// TwinCAT 3 PLC project PlcHammer
// Title: PlcHammer
// Company: Vortex.Library
// ProjectVersion: 0.6.0.913
// ProgramVersion: 3.1.4023.0
// libraries:
//   Tc2_Math, * (Beckhoff Automation GmbH)
//   Tc2_Standard, * (Beckhoff Automation GmbH)
//   Tc2_System, * (Beckhoff Automation GmbH)
//   Tc3_Module, * (Beckhoff Automation GmbH)
//   TcoCore, 0.8.1.3 (Vortex.Library)
//   TcoData, 0.8.1.3 (Vortex.Library)
//   TcoDrivesBeckhoff, 0.8.1.3 (Vortex.Library)
//   TcoElements, 0.8.1.3 (Vortex.Library)
//   TcoInspectors, 0.6.0.913 (Vortex.Library)
//   TcoIo, 0.8.1.3 (Vortex.Library)
//   TcoPneumatics, 0.8.1.3 (Vortex.Library)
// project tree:
//   Components/Drive/ DriveSim.TcPOU (not stored), DriveSimMoveAbsoluteTask.TcPOU (not stored), IDrive.TcIO (not stored)
//   DUTs/Enums/ enumColors.TcDUT, enumModes.TcDUT (not stored)
//   DUTs/Structs/CutomLibraries/ VortexComponent.TcDUT
//   DUTs/Structs/GenericStructs/ Car.TcDUT, VariousTypes.TcDUT, Wheel.TcDUT
//   DUTs/Structs/LayoutTests/Border/ BorderLayout.TcDUT, Border_other.TcDUT
//   DUTs/Structs/LayoutTests/GroupBox/ GroupBoxLayout.TcDUT, GroupBox_other.TcDUT
//   DUTs/Structs/LayoutTests/Multiple/ Border_other_other.TcDUT, GroupBox_other_other.TcDUT, Scroll_other_other.TcDUT, Stack_other_other.TcDUT, Tabs_other_other.TcDUT, UniformGrid_other_other.TcDUT, Wrap_other_other.TcDUT
//   DUTs/Structs/LayoutTests/Scroll/ ScrollLayout.TcDUT, Scroll_other.TcDUT
//   DUTs/Structs/LayoutTests/Stack/ StackLayout.TcDUT, Stack_other.TcDUT
//   DUTs/Structs/LayoutTests/Tabs/ TabsLayout.TcDUT (not stored), Tabs_other.TcDUT
//   DUTs/Structs/LayoutTests/UniformGrid/ UniformGridLayout.TcDUT, UniformGrid_other.TcDUT
//   DUTs/Structs/ LayoutTests.TcDUT, RenderIgnoreTests.TcDUT
//   DUTs/Structs/LayoutTests/Wrap/ WrapLayout.TcDUT (not stored), Wrap_other.TcDUT
//   DUTs/Structs/RenderIgnore/ RenderIgnore_basic.TcDUT
//   Misc/Checkers/ Checkers.TcPOU (not stored), AnalogueValueCheck.TcDUT (not stored), eCheckResult.TcDUT (not stored)
//   / PlcTask.TcTTO (not stored)
//   POUs/ AppContext.TcPOU (not stored), TECH_MAIN.TcPOU (not stored)
//   POUs/Data/ ProcessDataManager.TcPOU (not stored), RealValueSimulation.TcPOU (not stored), TechnologicalDataManager.TcPOU (not stored)
//   POUs/Station001/ Station001_Swift.TcPOU (not stored), IO.TcGVL (not stored), Station001.TcPOU, Station001_Components.TcPOU (not stored), Station001_GroundMode.TcPOU (not stored), Station001_AutomatMode.TcPOU (not stored), Station001_ProductionData.TcDUT (not stored), Station001_TechnologicalSettings.TcDUT (not stored)
// real-time tasks:
//   TASK PlcTask: cycle T#10ms, priority 20, ADS port 350
// motion (NC):
//   TASK NC-Task 1 SAF: cycle T#2ms, priority 4, ADS port 501
//   TASK NC-Task 1 SVB: cycle T#10ms, priority 8, ADS port 511
//   AXIS Axis 1 (id 1)
//     OtherSettings: AllowMotionCmdToSlave=true
//     encoder EncType=1
//     drive DrvType=5
//       Analog: TorqueSetpointScale=10, ScaleFactorActTorque=0.1
//       TimeComp: TaskDelayCycles=1
//     controller CtrType=1
//       CtrPara: PriorControlFactor=1
//         Observer: BandWidth=20
// variable links:
//   PlcHammer/PlcHammer Instance <-> NC-Task 1 SAF/Axes/Axis 1
//     PlcTask Inputs/IO.Axis1.NcToPlc <-> Outputs/ToPlc
//     PlcTask Outputs/IO.Axis1.PlcToNc <-> Inputs/FromPlc

// ---- DUTs/Enums/enumColors.TcDUT
{attribute 'qualified_only'}
{attribute 'strict'}
TYPE enumColors :
(
	Red := 0,
	Orange := 1,
	Yellow := 2,
	Green := 3,
	Blue := 4,
	Indigo := 5,
	Violet := 6
);
END_TYPE

// ---- DUTs/Structs/CutomLibraries/VortexComponent.TcDUT
TYPE VortexComponent :
STRUCT
	vortex_bool: BOOL;
	vortex_int: INT;
	vortex_string: STRING;
	vortex_wheel: Wheel;
END_STRUCT
END_TYPE

// ---- DUTs/Structs/GenericStructs/Car.TcDUT
TYPE Car :
STRUCT
	_manufacturer: STRING;
	_model: STRING;
	_manufactured_time: DATE_AND_TIME;
	_ready_for_UK: BOOL;
	_color: enumColors;
	_width: REAL;
	_height: REAL;
	_length: REAL;
	_price: USINT;
END_STRUCT
END_TYPE

// ---- DUTs/Structs/GenericStructs/VariousTypes.TcDUT
TYPE VariousTypes :
STRUCT
	_BOOL_00          : BOOL;
	_INT_00           : INT;
	{attribute addProperty Name "<#_UINT_00 with subrange 69-420#>"}
	_UINT_00          : UINT (69..420);
	_ULINT_00         : ULINT := 18446744073709551615;
	_REAL_00          : REAL := 2.718281828;
	_BYTE_00          : BYTE := 2#00000101;
	_DATE_AND_TIME_00 : DATE_AND_TIME := DT#2000-01-01-00:00:00.01;
	_LTIME_00         : LTIME := LTIME#2D0H45M1S563MS333US880NS;
	{attribute clr [RenderIgnore()]}
	_STRING_00        : STRING;
	_STRING_01        : STRING := 'How are you?';
	_ptString         : POINTER TO STRING := ADR(_STRING_01);
	_eColors_00       : enumColors := enumColors.Red;
END_STRUCT
END_TYPE

// ---- DUTs/Structs/GenericStructs/Wheel.TcDUT
TYPE Wheel :
STRUCT
	_rim_radius: REAL;
	_material: STRING;
	_manufactured_time: DATE_AND_TIME;
END_STRUCT
END_TYPE

// ---- DUTs/Structs/LayoutTests/Border/BorderLayout.TcDUT
{attribute wpf [Container(Layout.Border)]}
TYPE BorderLayout:
STRUCT
	_various_types: VariousTypes;
END_STRUCT
END_TYPE

// ---- DUTs/Structs/LayoutTests/Border/Border_other.TcDUT
{attribute wpf [Container(Layout.Border)]}
TYPE Border_other :
STRUCT
	{attribute wpf [Container(Layout.Stack)]}
	_wheel_stack: Wheel;
	{attribute wpf [Container(Layout.UniformGrid)]}
	_wheel_ug: Wheel;
	{attribute wpf [Container(Layout.Wrap)]}
	_wheel_wrap: Wheel;
	{attribute wpf [Container(Layout.Tabs)]}
	_wheel_tabs: Wheel;
	{attribute wpf [Container(Layout.Border)]}
	_wheel_border: Wheel;
	{attribute wpf [Container(Layout.GroupBox)]}
	_wheel_gb: Wheel;
	{attribute wpf [Container(Layout.Scroll)]}
	_wheel_scroll: Wheel;
END_STRUCT
END_TYPE

// ---- DUTs/Structs/LayoutTests/GroupBox/GroupBoxLayout.TcDUT
TYPE GroupBoxLayout:
STRUCT
	{attribute wpf [Container(Layout.Stack)]}
	{attribute wpf [Group(Layout.GroupBox)]}
	{attribute addProperty Name "<#Various types#>"}
	_vt: VariousTypes;
END_STRUCT
END_TYPE

// ---- DUTs/Structs/LayoutTests/GroupBox/GroupBox_other.TcDUT
{attribute wpf [Container(Layout.GroupBox)]}
TYPE GroupBox_other :
STRUCT
	{attribute wpf [Container(Layout.Stack)]}
	_wheel_stack: Wheel;
	{attribute wpf [Container(Layout.UniformGrid)]}
	_wheel_ug: Wheel;
	{attribute wpf [Container(Layout.Wrap)]}
	_wheel_wrap: Wheel;
//	{attribute wpf [Container(Layout.Tabs)]}
//	_wheel_tabs: Wheel;
	{attribute wpf [Container(Layout.Border)]}
	_wheel_border: Wheel;
	{attribute wpf [Container(Layout.Scroll)]}
	_wheel_scroll: Wheel;
END_STRUCT
END_TYPE

// ---- DUTs/Structs/LayoutTests/Multiple/Border_other_other.TcDUT
{attribute wpf [Container(Layout.Border)]}
TYPE Border_other_other :
STRUCT
	{attribute addProperty Name "<#Stack#>"}
	_stack_other: Stack_other;
	{attribute addProperty Name "<#UniformGrid#>"}
	_uniformGrid_other: UniformGrid_other;
	{attribute addProperty Name "<#Wrap#>"}
	_wrap_other: Wrap_other;
	{attribute addProperty Name "<#Tabs#>"}
	_tabs_other: Tabs_other;
	{attribute addProperty Name "<#Border#>"}
	_border_other: Border_other;
	{attribute addProperty Name "<#GroupBox#>"}
	_groupBox_other: GroupBox_other;
	{attribute addProperty Name "<#Scroll#>"}
	_scroll_other: Scroll_other;
END_STRUCT
END_TYPE

// ---- DUTs/Structs/LayoutTests/Multiple/GroupBox_other_other.TcDUT
{attribute wpf [Container(Layout.GroupBox)]}
TYPE GroupBox_other_other :
STRUCT
	{attribute addProperty Name "<#Stack#>"}
	_stack_other: Stack_other;
	{attribute addProperty Name "<#UniformGrid#>"}
	_uniformGrid_other: UniformGrid_other;
	{attribute addProperty Name "<#Wrap#>"}
	_wrap_other: Wrap_other;
	{attribute addProperty Name "<#Tabs#>"}
	_tabs_other: Tabs_other;
	{attribute addProperty Name "<#Border#>"}
	_border_other: Border_other;
	{attribute addProperty Name "<#GroupBox#>"}
	_groupBox_other: GroupBox_other;
	{attribute addProperty Name "<#Scroll#>"}
	_scroll_other: Scroll_other;
END_STRUCT
END_TYPE

// ---- DUTs/Structs/LayoutTests/Multiple/Scroll_other_other.TcDUT
{attribute wpf [Container(Layout.Scroll)]}
TYPE Scroll_other_other :
STRUCT
	{attribute addProperty Name "<#Stack#>"}
	_stack_other: Stack_other;
	{attribute addProperty Name "<#UniformGrid#>"}
	_uniformGrid_other: UniformGrid_other;
	{attribute addProperty Name "<#Wrap#>"}
	_wrap_other: Wrap_other;
	{attribute addProperty Name "<#Tabs#>"}
	_tabs_other: Tabs_other;
	{attribute addProperty Name "<#Border#>"}
	_border_other: Border_other;
	{attribute addProperty Name "<#GroupBox#>"}
	_groupBox_other: GroupBox_other;
	{attribute addProperty Name "<#Scroll#>"}
	_scroll_other: Scroll_other;
END_STRUCT
END_TYPE

// ---- DUTs/Structs/LayoutTests/Multiple/Stack_other_other.TcDUT
{attribute wpf [Container(Layout.Stack)]}
TYPE Stack_other_other :
STRUCT
	{attribute addProperty Name "<#Stack#>"}
	_stack_other: Stack_other;
	{attribute addProperty Name "<#UniformGrid#>"}
	_uniformGrid_other: UniformGrid_other;
	{attribute addProperty Name "<#Wrap#>"}
	_wrap_other: Wrap_other;
	{attribute addProperty Name "<#Tabs#>"}
	_tabs_other: Tabs_other;
	{attribute addProperty Name "<#Border#>"}
	_border_other: Border_other;
	{attribute addProperty Name "<#GroupBox#>"}
	_groupBox_other: GroupBox_other;
	{attribute addProperty Name "<#Scroll#>"}
	_scroll_other: Scroll_other;
END_STRUCT
END_TYPE

// ---- DUTs/Structs/LayoutTests/Multiple/Tabs_other_other.TcDUT
{attribute wpf [Container(Layout.Tabs)]}
TYPE Tabs_other_other :
STRUCT
	{attribute addProperty Name "<#Stack#>"}
	_stack_other: Stack_other;
	{attribute addProperty Name "<#UniformGrid#>"}
	_uniformGrid_other: UniformGrid_other;
	{attribute addProperty Name "<#Wrap#>"}
	_wrap_other: Wrap_other;
	{attribute addProperty Name "<#Tabs#>"}
	_tabs_other: Tabs_other;
	{attribute addProperty Name "<#Border#>"}
	_border_other: Border_other;
	{attribute addProperty Name "<#GroupBox#>"}
	_groupBox_other: GroupBox_other;
	{attribute addProperty Name "<#Scroll#>"}
	_scroll_other: Scroll_other;
END_STRUCT
END_TYPE

// ---- DUTs/Structs/LayoutTests/Multiple/UniformGrid_other_other.TcDUT
{attribute wpf [Container(Layout.UniformGrid)]}
TYPE UniformGrid_other_other :
STRUCT
	{attribute addProperty Name "<#Stack#>"}
	_stack_other: Stack_other;
	{attribute addProperty Name "<#UniformGrid#>"}
	_uniformGrid_other: UniformGrid_other;
	{attribute addProperty Name "<#Wrap#>"}
	_wrap_other: Wrap_other;
	{attribute addProperty Name "<#Tabs#>"}
	_tabs_other: Tabs_other;
	{attribute addProperty Name "<#Border#>"}
	_border_other: Border_other;
	{attribute addProperty Name "<#GroupBox#>"}
	_groupBox_other: GroupBox_other;
	{attribute addProperty Name "<#Scroll#>"}
	_scroll_other: Scroll_other;
END_STRUCT
END_TYPE

// ---- DUTs/Structs/LayoutTests/Multiple/Wrap_other_other.TcDUT
{attribute wpf [Container(Layout.Wrap)]}
TYPE Wrap_other_other :
STRUCT
	{attribute addProperty Name "<#Stack#>"}
	_stack_other: Stack_other;
	{attribute addProperty Name "<#UniformGrid#>"}
	_uniformGrid_other: UniformGrid_other;
	{attribute addProperty Name "<#Wrap#>"}
	_wrap_other: Wrap_other;
	{attribute addProperty Name "<#Tabs#>"}
	_tabs_other: Tabs_other;
	{attribute addProperty Name "<#Border#>"}
	_border_other: Border_other;
	{attribute addProperty Name "<#GroupBox#>"}
	_groupBox_other: GroupBox_other;
	{attribute addProperty Name "<#Scroll#>"}
	_scroll_other: Scroll_other;
END_STRUCT
END_TYPE

// ---- DUTs/Structs/LayoutTests/Scroll/ScrollLayout.TcDUT
{attribute wpf [Container(Layout.Scroll)]}
TYPE ScrollLayout :
STRUCT
	_vt: VariousTypes;
END_STRUCT
END_TYPE

// ---- DUTs/Structs/LayoutTests/Scroll/Scroll_other.TcDUT
{attribute wpf [Container(Layout.Scroll)]}
TYPE Scroll_other :
STRUCT
	{attribute wpf [Container(Layout.Stack)]}
	_wheel_stack: Wheel;
	{attribute wpf [Container(Layout.UniformGrid)]}
	_wheel_ug: Wheel;
	{attribute wpf [Container(Layout.Wrap)]}
	_wheel_wrap: Wheel;
	{attribute wpf [Container(Layout.Tabs)]}
	_wheel_tabs: Wheel;
	{attribute wpf [Container(Layout.Border)]}
	_wheel_border: Wheel;
	{attribute wpf [Container(Layout.GroupBox)]}
	_wheel_gb: Wheel;
	{attribute wpf [Container(Layout.Scroll)]}
	_wheel_scroll: Wheel;
END_STRUCT
END_TYPE

// ---- DUTs/Structs/LayoutTests/Stack/StackLayout.TcDUT
{attribute wpf [Container(Layout.Stack)]}
TYPE StackLayout:
STRUCT
	_various_types: VariousTypes;
END_STRUCT
END_TYPE

// ---- DUTs/Structs/LayoutTests/Stack/Stack_other.TcDUT
{attribute wpf [Container(Layout.Stack)]}
TYPE Stack_other :
STRUCT
	{attribute wpf [Container(Layout.Stack)]}
	_wheel_stack: Wheel;
	{attribute wpf [Container(Layout.UniformGrid)]}
	_wheel_ug: Wheel;
	{attribute wpf [Container(Layout.Wrap)]}
	_wheel_wrap: Wheel;
	{attribute wpf [Container(Layout.Tabs)]}
	_wheel_tabs: Wheel;
	{attribute wpf [Container(Layout.Border)]}
	_wheel_border: Wheel;
	{attribute wpf [Container(Layout.GroupBox)]}
	_wheel_gb: Wheel;
	{attribute wpf [Container(Layout.Scroll)]}
	_wheel_scroll: Wheel;
END_STRUCT
END_TYPE

// ---- DUTs/Structs/LayoutTests/Tabs/Tabs_other.TcDUT
{attribute wpf [Container(Layout.Tabs)]}
TYPE Tabs_other :
STRUCT
	{attribute addProperty Name "<#Stack#>"}
	{attribute wpf [Container(Layout.Stack)]}
	_wheel_stack: Wheel;
	{attribute addProperty Name "<#UniformGrid#>"}
	{attribute wpf [Container(Layout.UniformGrid)]}
	_wheel_ug: Wheel;
	{attribute addProperty Name "<#Wrap#>"}
	{attribute wpf [Container(Layout.Wrap)]}
	_wheel_wrap: Wheel;
	{attribute addProperty Name "<#Tabs#>"}
	{attribute wpf [Container(Layout.Tabs)]}
	_wheel_tabs: Wheel;
	{attribute addProperty Name "<#Border#>"}
	{attribute wpf [Container(Layout.Border)]}
	_wheel_border: Wheel;
	{attribute addProperty Name "<#GroupBox#>"}
	{attribute wpf [Container(Layout.GroupBox)]}
	_wheel_gb: Wheel;
	{attribute addProperty Name "<#Scroll#>"}
	{attribute wpf [Container(Layout.Scroll)]}
	_wheel_scroll: Wheel;
END_STRUCT
END_TYPE

// ---- DUTs/Structs/LayoutTests/UniformGrid/UniformGridLayout.TcDUT
{attribute wpf [Container(Layout.UniformGrid)]}
TYPE UniformGridLayout:
STRUCT
	_various_types: VariousTypes;
END_STRUCT
END_TYPE

// ---- DUTs/Structs/LayoutTests.TcDUT
TYPE LayoutTests :
STRUCT
	_stackLayout: StackLayout;
	_uniformGridLayout: UniformGridLayout;
	_wrapLayout: WrapLayout;
	_tabsLayout: TabsLayout;
	_borderLayout: BorderLayout;
	_groupBoxLayout: GroupBoxLayout;
	_scrollLayout: ScrollLayout;
	
	// multiple 2nd layer
	_stack_other: Stack_other;
	_uniformGrid_other: UniformGrid_other;
	_wrap_other: Wrap_other;
	_tabs_other: Tabs_other;
	_border_other: Border_other;
	_groupBox_other: GroupBox_other;
	_scroll_other: Scroll_other;
	
	//multiple 3rd layer xddds
	_stack_other_other: Stack_other_other;
	_uniformGrid_other_other: UniformGrid_other_other;
	_wrap_other_other: Wrap_other_other;
	_tabs_other_other: Tabs_other_other;
	_border_other_other: Border_other_other;
	_groupBox_other_other: GroupBox_other_other;
	_scroll_other_other: Scroll_other_other;
END_STRUCT
END_TYPE

// ---- DUTs/Structs/LayoutTests/UniformGrid/UniformGrid_other.TcDUT
{attribute wpf [Container(Layout.UniformGrid)]}
TYPE UniformGrid_other :
STRUCT
	{attribute wpf [Container(Layout.Stack)]}
	_wheel_stack: Wheel;
	{attribute wpf [Container(Layout.UniformGrid)]}
	_wheel_ug: Wheel;
	{attribute wpf [Container(Layout.Wrap)]}
	_wheel_wrap: Wheel;
	{attribute wpf [Container(Layout.Tabs)]}
	_wheel_tabs: Wheel;
	{attribute wpf [Container(Layout.Border)]}
	_wheel_border: Wheel;
	{attribute wpf [Container(Layout.GroupBox)]}
	_wheel_gb: Wheel;
	{attribute wpf [Container(Layout.Scroll)]}
	_wheel_scroll: Wheel;
END_STRUCT
END_TYPE

// ---- DUTs/Structs/LayoutTests/Wrap/Wrap_other.TcDUT
{attribute wpf [Container(Layout.Wrap)]}
TYPE Wrap_other :
STRUCT
	{attribute wpf [Container(Layout.Stack)]}
	_wheel_stack: Wheel;
	{attribute wpf [Container(Layout.UniformGrid)]}
	_wheel_ug: Wheel;
	{attribute wpf [Container(Layout.Wrap)]}
	_wheel_wrap: Wheel;
	{attribute wpf [Container(Layout.Tabs)]}
	_wheel_tabs: Wheel;
	{attribute wpf [Container(Layout.Border)]}
	_wheel_border: Wheel;
	{attribute wpf [Container(Layout.GroupBox)]}
	_wheel_gb: Wheel;
	{attribute wpf [Container(Layout.Scroll)]}
	_wheel_scroll: Wheel;
END_STRUCT
END_TYPE

// ---- DUTs/Structs/RenderIgnoreTests.TcDUT
TYPE RenderIgnoreTests :
STRUCT
	_renderIgnore_basic: RenderIgnore_basic;
END_STRUCT
END_TYPE

// ---- DUTs/Structs/RenderIgnore/RenderIgnore_basic.TcDUT
TYPE RenderIgnore_basic :
STRUCT
	{attribute clr [RenderIgnore()]}
	_wheel_all: INT;
	
	{attribute clr [RenderIgnore("Display")]}
	_wheel_display: INT;
	
	{attribute clr [RenderIgnore("Control")]}
	_wheel_control: INT;
	
	{attribute clr [RenderIgnore("ShadowDisplay")]}
	_wheel_shadowDisplay: INT;
	
	{attribute clr [RenderIgnore("ShadowControl")]}
	_wheel_shadowControl: INT;
	
	//
	
	{attribute clr [RenderIgnore("ShadowControl", "ShadowDisplay")]}
	_wheel_sC_sD: INT;
	
	{attribute clr [RenderIgnore("Control", "Display")]}
	_wheel_C_D: INT;
	
	//
	
	{attribute clr [RenderIgnore("Control", "Display", "ShadowControl")]}
	_wheel_C_D_sC: INT;
END_STRUCT
END_TYPE

// ---- POUs/Station001/Station001.TcPOU
FUNCTION_BLOCK Station001 EXTENDS TcoCore.TcoObject 
VAR
	_components : Station001_Components(THIS^);
	
	_groundMode : Station001_GroundMode(THIS^, eRestoreMode.None);
	_automatMode : Station001_AutomatMode(THIS^, eRestoreMode.None);
	_swiftSequence   : Station001_Swift(THIS^, eRestoreMode.None);
	
	_groundModeTask : TcoCore.TcoTask(THIS^);
	_automatModeTask : TcoCore.TcoTask(THIS^);
	_serviceModeTask : TcoCore.TcoTask(THIS^);
	_swiftModeTask : TcoCore.TcoTask(THIS^);
	
	
	_processRecipies : ProcessDataManager(THIS^); 
    _processTraceabilty : ProcessDataManager(THIS^);
	_technologicalDataManager : TechnologicalDataManager(THIS^);
	_currentMode : enumModes := enumModes.Idle;
	_checkers : Checkers(THIS^);
	
	_layoutTests: LayoutTests;
	_renderIgnoreTests: RenderIgnoreTests;
	_vortexComponent: VortexComponent;
END_VAR

_components();
_processRecipies();
_processTraceabilty();
_technologicalDataManager();

ServiceMode();
GroundMode();
AutomatMode();


IF(_swiftModeTask.Execute()) THEN
	Messenger.Trace('Service mode active');	
	_automatModeTask.Restore();
	_groundModeTask.Restore();
	_groundMode.Restore();
	_automatMode.Restore();
	_serviceModeTask.Restore();
	_swiftSequence.Run();
	_currentMode := enumModes.Idle;
END_IF

METHOD AutomatMode : BOOL
VAR_INPUT
END_VAR
_automatModeTask.Enabled := _groundModeTask.Done;

IF(_automatModeTask.Execute()) THEN
	Messenger.Trace('Automat mode active');
	_serviceModeTask.Abort();
	_automatMode.Run();
	_currentMode := enumModes.Automat;
END_IF
END_METHOD

PROPERTY Checkers : REFERENCE TO Checkers
GET
Checkers REF= _checkers;
END_GET
END_PROPERTY

PROPERTY Components : REFERENCE TO Station001_Components
GET
Components REF= _components;
END_GET
END_PROPERTY

METHOD GroundMode : BOOL
VAR_INPUT
END_VAR
IF(_groundModeTask.Execute()) THEN
	Messenger.Trace('Ground position mode active');
	_serviceModeTask.Restore();
	_automatModeTask.Restore();
	_automatMode.Restore();
	_groundMode.Run();
	_groundModeTask.DoneWhen(_groundMode.CurrentStep.ID = 300);
	IF _groundModeTask.Done THEN
		_groundMode.Restore();
	END_IF
	_currentMode := enumModes.Ground;
END_IF
END_METHOD

PROPERTY ProcessRecepie : REFERENCE TO ProcessDataManager
GET
ProcessRecepie REF= _processRecipies;
END_GET
END_PROPERTY

PROPERTY ProcessTraceabilty : REFERENCE TO ProcessDataManager
GET
ProcessTraceabilty REF= _processTraceabilty;
END_GET
END_PROPERTY

PROPERTY  ProductionData : REFERENCE TO Station001_ProductionData
GET
ProductionData REF= _processTraceabilty._data;
END_GET
END_PROPERTY

METHOD ServiceMode
VAR_INPUT
END_VAR
IF(_serviceModeTask.Execute()) THEN
	Messenger.Trace('Service mode active');	
	_automatModeTask.Restore();
	_groundModeTask.Restore();
	_groundMode.Restore();
	_automatMode.Restore();
	_components.Service();
	_currentMode := enumModes.Service;
END_IF
END_METHOD

PROPERTY TechnologicalDataManager : REFERENCE TO TechnologicalDataManager
GET
TechnologicalDataManager REF= _technologicalDataManager;
END_GET
END_PROPERTY

END_FUNCTION_BLOCK
